{attribute 'qualified_only'}
{attribute 'strict'}
TYPE cPuckStatusEval :
(
	
	None := 0

) DINT;
END_TYPE

(* stored: Version 1.1.0.1, ProductVersion 3.1.4024.6
   DUT cPuckStatusEval: Id {55cf5f27-c399-45b6-81a8-0b445482c478} *)
